(* CODESYS project TrafficLight.project

Project tree, tasks and I/O mapping:
  Device : CODESYS Control Win V3, 3S - Smart Software Solutions GmbH, order no. 305021, version 3.5.5.50
    application Application
      libraries: Standard, * (System); MQTT Client Library, 3.5.13.20 (Stefan Roßmann Engineering Solutions)
      task MainTask (cyclic, interval t#20ms, priority 1) calls PLC_PRG
      program PLC_PRG [CFC]
*)

// Device/Application/PLC_PRG
PROGRAM PLC_PRG
VAR
	MQTT_Client_FB_MQTTClient_1 : MQTT_Client.FB_MQTTClient;
	xSub: BOOL := true;
END_VAR

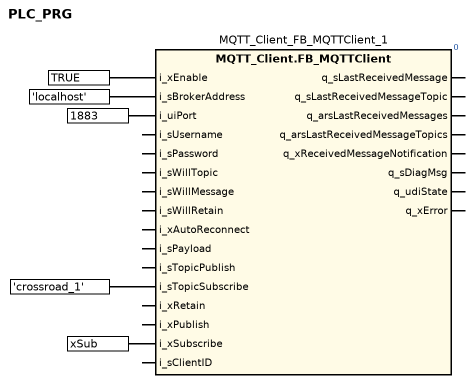
MQTT_Client_FB_MQTTClient_1(
    i_xEnable := TRUE,
    i_sBrokerAddress := 'localhost',
    i_uiPort := 1883,
    i_sTopicSubscribe := 'crossroad_1',
    i_xSubscribe := xSub); // MQTT_Client.FB_MQTTClient

END_PROGRAM
